FUNCTION_BLOCK FB_OtherThing
VAR_INPUT
END_VAR
VAR_OUTPUT
END_VAR
VAR
	counter	: INT; 
END_VAR

counter := counter + 1

METHOD DoSomething : BOOL
VAR_INPUT
END_VAR
counter := counter + 1
END_METHOD

END_FUNCTION_BLOCK

(* stored: Version 1.1.0.1, ProductVersion 3.1.4024.0
   POU FB_OtherThing: Id {ab3294b6-c055-49d9-b8f7-44f33997f393}, SpecialFunc None
   Method DoSomething: Id {b8c1536c-55ed-4d75-80ed-bc5144d16344} *)
